// TIA Portal V18 export
TYPE "LGasp_typeArticoloGenerale"
// stored: IsFailsafeCompliant false
   STRUCT
      "name" : WString[30];   // nome dell'articolo
      lenght : LReal := -1.0;   // [mm] - Lunghezza totale npezzi + sfrido (eventuale)
      nominal_lenght : LReal := -1.0;   // [mm] - lunghezza nominale per gestione pezzi non multipli dello stampo / [mm] - Lunghezza dei pezzi non multipli del passo del feeder
      cutoffset : LReal := -1.0;   // [mm] - Offset foro sincronismo - taglio (eventuale)
      options : Array[1..16] of Bool;   // disponibile per opzioni varie
      options_str : Array[1..3] of WString[20];   // disponibile per dati specifici dell'impianto
      options_lreal : Array[1..3] of LReal;   // disponibile per dati specifici dell'impianto
      options_dint : Array[1..3] of DInt;   // disponibile per dati specifici dell'impianto
      print { S7_SetPoint := 'True'} : "LGasp_typeStampante";
   END_STRUCT;
   // // options[1] : Taglio con ruota metrica (0: No, 1: Si)
   // // options[2] : Articolo rastremato (0: No, 1: Si)
   // // options[3] : Prodotto NON forato (0: pz forato, 1: pz non forato)
   // // options[4] : Taglio con oscuramento (1: abilitato)
   // // options[5] : Panno anticondensa
   // // options[6] : Film protettivo pelabile 1 (lato superiore)
   // // options[7] : Film protettivo pelabile 2 (lato inferiore)
   // // options[8] : pacco con 0=listelli+tavola 1=listelli+listelli
   // // options[16] : Scarto per giunzione (0: pz ok, 1: pz scarto)
END_TYPE
